PROGRAM MAIN
VAR
	iCount:INT;
	bStart:BOOL;
	bTestVar:BOOL;
END_VAR

IF bStart THEN
	iCount := iCount+1;
ELSE
	iCount := 0;
END_IF

END_PROGRAM

(* stored: Version 1.1.0.1, ProductVersion 3.1.4024.9
   POU MAIN: Id {1f1ae45e-71c9-478c-97b0-d7f07dab23e5}, SpecialFunc None *)
